TYPE ST_Nest :
STRUCT
    nId                       : UINT;
    ePosition                 : E_TablePosition;
    bEnabled                  : BOOL;
    bPartPresent              : BOOL;
    bPreviousPartPresent      : BOOL;
    bPartLoadedPulse          : BOOL;
    bPartRemovedPulse         : BOOL;
    bProcessRequired          : BOOL;
    bProcessComplete          : BOOL;
    eDisposition              : E_PartDisposition;
    bDispositionSent          : BOOL;
    bOperatorExchangeComplete : BOOL;
    stPatchDispenseResult     : ST_ProcessResult;
    stHeatStakeResult         : ST_ProcessResult;
    stVisionResult            : ST_ProcessResult;
    stResult                  : ST_ProcessResult;
    bStatisticsCounted        : BOOL;
END_STRUCT
END_TYPE

(* stored: Version 1.1.0.1, ProductVersion 3.1.4026.18
   DUT ST_Nest: Id {e9c52966-abb7-45b8-ba6f-050cecbcb7e1} *)
